FUNCTION_BLOCK threshold (* openCV threshold *)
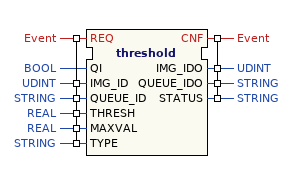
  EVENT_INPUT
    REQ WITH IMG_ID, QUEUE_ID, THRESH, MAXVAL, TYPE;
  END_EVENT
  EVENT_OUTPUT
    CNF WITH IMG_IDO, QUEUE_IDO, STATUS;
  END_EVENT
  VAR_INPUT
    QI : BOOL;
    IMG_ID : UDINT;
    QUEUE_ID : STRING;
    THRESH : REAL;
    MAXVAL : REAL;
    TYPE : STRING;
  END_VAR
  VAR_OUTPUT
    IMG_IDO : UDINT;
    QUEUE_IDO : STRING;
    STATUS : STRING;
  END_VAR
END_FUNCTION_BLOCK
